// TIA Portal project "Proyecto 4" (V17)
// Clasificador de Cajas

(* hardware
DEVICE "S7-1500/ET200MP station_1"  S7-1500 station
   slot 0: "Rail_0"  Rack  6ES7 590-1***0-0AA0
   slot 1: "PLC_1"  CPU 1515-2 PN  6ES7 515-2AM02-0AB0  V2.9
      slot 3: "CPU display_1"  6ES7591-1BA00-0AA0
      slot 32768: "PROFINET interface_1"  X1
         slot 32769: "Port_1"  X1 P1
         slot 32770: "Port_2"  X1 P2
      slot 33024: "PROFINET interface_2"  X2
         slot 33025: "Port_1"  X2 P1
      slot 34817: "Virtual CP interface port_1"  Virtual CP interface port  Virtual CP interface port
   slot 2: "AI 8xU/I/RTD/TC ST_1"  AI 8xU/I/RTD/TC ST  6ES7 531-7KF00-0AB0  V2.0
   slot 3: "AI 8xU/I/RTD/TC ST_2"  AI 8xU/I/RTD/TC ST  6ES7 531-7KF00-0AB0  V2.0
   slot 4: "AI 8xU/I/RTD/TC ST_3"  AI 8xU/I/RTD/TC ST  6ES7 531-7KF00-0AB0  V2.0
   slot 5: "AI 8xU/I/RTD/TC ST_4"  AI 8xU/I/RTD/TC ST  6ES7 531-7KF00-0AB0  V2.0
   slot 6: "DI 16x24VDC BA_1"  DI 16x24VDC BA  6ES7 521-1BH10-0AA0  V1.0
*)

// ===== PLC "PLC_1"  CPU 1515-2 PN =====

VAR_GLOBAL   // PLC tag table "ED"
   "LAE-High" AT %I0.0 : Bool;
   "LAE-Low" AT %I0.1 : Bool;
   "LAE-Pallet" AT %I0.2 : Bool;
   "SLEN" AT %I0.3 : Bool;
   "SREN" AT %I0.4 : Bool;
   "SLEX" AT %I0.5 : Bool;
   "SREX" AT %I0.6 : Bool;
   "Marcha" AT %I0.7 : Bool;
   "Paro" AT %I1.0 : Bool;
   "Reset" AT %I1.1 : Bool;
   "Seta Emergencia" AT %I1.2 : Bool;
   "SL" AT %I1.3 : Bool;
   "Manual" AT %I1.4 : Bool;
   "Auto" AT %I1.5 : Bool;
END_VAR

VAR_GLOBAL   // PLC tag table "SD"
   "CT-right" AT %Q0.0 : Bool;
   "CT-left" AT %Q0.1 : Bool;
   "CT-Unload" AT %Q0.2 : Bool;
   "CT-Load" AT %Q0.3 : Bool;
   "CE" AT %Q0.4 : Bool;
   "CL" AT %Q0.5 : Bool;
   "CR" AT %Q0.6 : Bool;
   "Emitter" AT %Q0.7 : Bool;
   "Remover left" AT %Q1.0 : Bool;
   "Remover right" AT %Q1.1 : Bool;
   "Start light" AT %Q1.2 : Bool;
   "Stop light" AT %Q1.3 : Bool;
   "Reset light" AT %Q1.4 : Bool;
END_VAR

TYPE "UDT_Cinta"
   STRUCT
      Entradas : Struct
         ParoxSeguridad : Bool;
         Termico : Bool;
         Disyuntor : Bool;
         Auto : Bool;
         ConfMarcha : Bool;
         FalloVariador : Bool;
      END_STRUCT;
      Habilitado : Bool;
      Rearme : Bool;
      HMI : Struct
         Habilitado : Bool;
         segTrabajo : Int;
         minTrabajo : Int;
         horaTrabajo : Int;
      END_STRUCT;
      Alarma : Array[1..16] of Bool;
      AutoRearme : Array[1..16] of Bool;
      TimerAlarma : Array[1..16] of TON_TIME;
      TiempoAlarma : Array[1..16] of Time;
      "Timer" : Array[1..16] of TON_TIME;
      TimerON : Array[1..16] of Bool;
      Salidas : Struct
         Marcha : Bool;
      END_STRUCT;
      Permiso : Struct
         Externo : Bool;
      END_STRUCT;
   END_STRUCT;
END_TYPE

TYPE "UDT_Temporizador"
   STRUCT
      Congelacion : Bool;
      Reset : Bool;
      Q : Bool;
      Tiempo : Int;
      Conteo : Int;
   END_STRUCT;
END_TYPE

TYPE "UDT_Sensor"
   STRUCT
      Value : Bool;
      TON : "UDT_Temporizador";
   END_STRUCT;
END_TYPE

TYPE "UDT_Cinta_Bilateral"
   STRUCT
      Entradas : Struct
         ParoxSeguridad : Bool;
         Termico : Bool;
         Disyuntor : Bool;
         Auto : Bool;
         ConfMarcha : Bool;
         FalloVariador : Bool;
      END_STRUCT;
      Habilitado : Bool;
      Rearme : Bool;
      HMI : Struct
         Habilitado : Bool;
         segTrabajo : Int;
         minTrabajo : Int;
         horaTrabajo : Int;
      END_STRUCT;
      Alarma : Array[1..16] of Bool;
      AutoRearme : Array[1..16] of Bool;
      TimerAlarma : Array[1..16] of TON_TIME;
      TiempoAlarma : Array[1..16] of Time;
      "Timer" : Array[1..16] of TON_TIME;
      TimerON : Array[1..16] of Bool;
      Salidas : Struct
         MarchaAdelante : Bool;
         MarchaAtras : Bool;
         MarchaDch : Bool;
         MarchaIzq : Bool;
      END_STRUCT;
      Permiso : Struct
         Adelante : Bool;
         Atras : Bool;
         Derecha : Bool;
         Izquierda : Bool;
      END_STRUCT;
   END_STRUCT;
END_TYPE

DATA_BLOCK "DB_Generalidades"   // DB1
{ S7_Optimized_Access := 'TRUE' }
VERSION : 0.1
   VAR
      SiempreON : Bool;
      SiempreOFF : Bool;
      Tiempo : Struct
         Imp1ms : Bool;
         Imp1s : Bool;
         Imp1m : Bool;
         Imp1h : Bool;
         TON1ms : TON_TIME;
         TON1s : TON_TIME;
         TON1m : TON_TIME;
         TON1h : TON_TIME;
      END_STRUCT;
   END_VAR
BEGIN
END_DATA_BLOCK

// folder: 01_E/S

DATA_BLOCK "ED"   // DB2
{ S7_Optimized_Access := 'TRUE' }
VERSION : 0.1
   VAR
      "LAE-High" : Bool;
      "LAE-Low" : Bool;
      "LAE-Pallet" : Bool;
      SLEN : Bool;
      SREN : Bool;
      SLEX : Bool;
      SREX : Bool;
      Marcha : Bool;
      Paro : Bool;
      Reset : Bool;
      "Seta Emergencia" : Bool;
      SL : Bool;
      Manual : Bool;
      Auto : Bool;
   END_VAR
BEGIN
END_DATA_BLOCK

DATA_BLOCK "SD"   // DB3
{ S7_Optimized_Access := 'TRUE' }
VERSION : 0.1
   VAR
      "CT-right" : Bool;
      "CT-left" : Bool;
      "CT-Unload" : Bool;
      "CT-Load" : Bool;
      CE : Bool;
      CL : Bool;
      CR : Bool;
      Emitter : Bool;
      "Remover left" : Bool;
      "Remover right" : Bool;
      "Start light" : Bool;
      "Stop light" : Bool;
      "Reset light" : Bool;
   END_VAR
BEGIN
END_DATA_BLOCK

// folder: 02_Equipos

DATA_BLOCK "DB_SensoresDigitales"   // DB100
{ S7_Optimized_Access := 'TRUE' }
VERSION : 0.1
   VAR
      "LAE-High" : "UDT_Sensor";
      "LAE-Low" : "UDT_Sensor";
      "LAE-Pallet" : "UDT_Sensor";
      SLEN : "UDT_Sensor";
      SREN : "UDT_Sensor";
      SREX : "UDT_Sensor";
      SLEX : "UDT_Sensor";
      SetaEmergencia : "UDT_Sensor";
      SL : "UDT_Sensor";
      Paro : "UDT_Sensor";
   END_VAR
BEGIN
END_DATA_BLOCK

DATA_BLOCK "DB_Cintas"   // DB101
{ S7_Optimized_Access := 'TRUE' }
VERSION : 0.1
   VAR
      Unidireccional : Struct
         CE : "UDT_Cinta";
         CL : "UDT_Cinta";
         CR : "UDT_Cinta";
      END_STRUCT;
      Bidireccional : Struct
         CT : "UDT_Cinta_Bilateral";
      END_STRUCT;
   END_VAR
BEGIN
END_DATA_BLOCK

// folder: 10_Zona de Clasificacion

DATA_BLOCK "DB_ZonaClasificacion"   // DB200
{ S7_Optimized_Access := 'TRUE' }
VERSION : 0.1
   VAR
      EnMarcha : Bool;
      EnParo : Bool;
      Flanco : Array[1..32] of Bool;
      CajaEsperando : Bool;
      CajaEnCT : Bool;
      CajaGrande : Bool;
      CajaPequeña : Bool;
      CajaEnCR : Bool;
      CajaEnCL : Bool;
      CajasEnCR : Int;
      CajasEnCL : Int;
   END_VAR
BEGIN
END_DATA_BLOCK

// folder: (top level)

FUNCTION "FC_Generalidades" : Void   // FC1, LAD
{ S7_Optimized_Access := 'TRUE' }
VERSION : 0.1
BEGIN

REGION Network 1: +++++|SIEMPRE ON|+++++
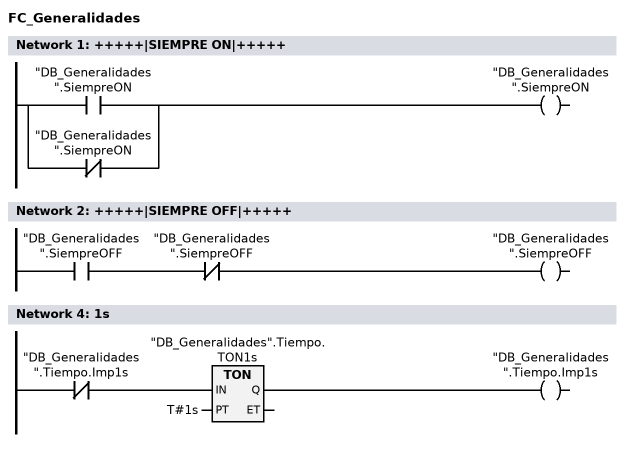
   RUNG wire#powerrail
      Contact( "DB_Generalidades".SiempreON )
      wire#w1
      Coil( "DB_Generalidades".SiempreON )
   END_RUNG
   RUNG wire#powerrail
      I_Contact( "DB_Generalidades".SiempreON )
   END_RUNG wire#w1
   // the same network as SCL:
   "DB_Generalidades".SiempreON := "DB_Generalidades".SiempreON OR NOT "DB_Generalidades".SiempreON;
END_REGION

REGION Network 2: +++++|SIEMPRE OFF|+++++
   RUNG wire#powerrail
      Contact( "DB_Generalidades".SiempreOFF )
      I_Contact( "DB_Generalidades".SiempreOFF )
      Coil( "DB_Generalidades".SiempreOFF )
   END_RUNG
   // the same network as SCL:
   "DB_Generalidades".SiempreOFF := "DB_Generalidades".SiempreOFF AND NOT "DB_Generalidades".SiempreOFF;
END_REGION

REGION Network 3: +++++|IMPULSOS DE TIEMPO|+++++
END_REGION

REGION Network 4: 1s
   "DB_Generalidades".Tiempo.TON1s.TON(IN := NOT "DB_Generalidades".Tiempo.Imp1s, PT := T#1s);
   "DB_Generalidades".Tiempo.Imp1s := "DB_Generalidades".Tiempo.TON1s.Q;
END_REGION
END_FUNCTION

FUNCTION "MHJ-PLC-Lab-Function-S71500" : Void   // FC9000, SCL
{ S7_Optimized_Access := 'TRUE' }
VERSION : 0.1
   VAR_TEMP
      Value : Byte;
      ForCounter : Int;
   END_VAR
   VAR CONSTANT
      Value_01_DW : DWord := 16#1223_5486;
      Value_02_DW : DWord := 16#A6C9_D1F5;
   END_VAR
BEGIN

   #Value:=PEEK(area := 16#82,
        dbNumber := 0,
        byteOffset := 511);
   #Value := #Value + 1;

   POKE(area := 16#82,
        dbNumber := 0,
        byteOffset := 511,
        value := #Value);

   POKE(area := 16#82,
        dbNumber := 0,
        byteOffset := 1016,
        value := #Value_01_DW);
   POKE(area := 16#82,
        dbNumber := 0,
        byteOffset := 1020,
        value := #Value_02_DW);

   FOR #ForCounter := 0 TO 63 DO
       #Value:=PEEK(area := 16#1,
            dbNumber := 0,
            byteOffset := #ForCounter);
       POKE(area := 16#81,
            dbNumber := 0,
            byteOffset := #ForCounter,
            value := #Value);
   END_FOR;
   #Value := PEEK(area := 16#1,
                  dbNumber := 0,
                  byteOffset := 512);
   POKE(area := 16#82,
        dbNumber := 0,
        byteOffset := 512,
        value := #Value);
END_FUNCTION

ORGANIZATION_BLOCK "Main"   // OB1, LAD, ProgramCycle
TITLE = "Main Program Sweep (Cycle)"
{ S7_Optimized_Access := 'TRUE' }
VERSION : 0.1
// BENONI BENJAMIN QUEZADA FLORES
   VAR_INPUT
      Initial_Call : Bool;   // Initial call of this OB
      Remanence : Bool;   // =True, if remanent data are available
   END_VAR
BEGIN

REGION Network 1 (STL): +++++|LECTURA ENTRADAS|+++++

         CALL  "FC_ED";
END_REGION

REGION Network 2 (STL): +++++|GENERALIDADES|+++++

         CALL  "FC_Generalidades";
END_REGION

REGION Network 3 (STL): +++++|COMUNICACION FACTORY IO|+++++

         CALL  "MHJ-PLC-Lab-Function-S71500";
END_REGION

REGION Network 4 (STL): +++++|ZONA CLASIFICACION|+++++

         CALL  "FC_ZonaClasificacion";
END_REGION

REGION Network 5 (STL): +++++|ESCRITURAS SALIDAS|+++++

         CALL  "FC_SD";
END_REGION
END_ORGANIZATION_BLOCK

// folder: 00_Bloques Estandar/FB

FUNCTION_BLOCK "FB_Motor"   // FB1, LAD
{ S7_Optimized_Access := 'TRUE' }
VERSION : 0.1
   VAR_INPUT
      eParoXSeguridad : Bool;
      eTermico : Bool;
      eDisyuntor : Bool;
      eAuto : Bool;
      eConfMarcha : Bool;
      eFalloVariador : Bool;
   END_VAR
   VAR_OUTPUT
      sMarcha : Bool;
   END_VAR
   VAR
      Habilitado : Bool;
      Rearme : Bool;
      PermisoExterno : Bool;
      HMI : Struct
         Habilitado : Bool;
         segTrabajo : Int;
         minTrabajo : Int;
         horaTrabajo : Int;
      END_STRUCT;
      Alarma : Array[1..16] of Bool;
      AutoRearme : Array[1..16] of Bool;
      TimerAlarma : Array[1..16] of TON_TIME;
      TiempoAlarma : Array[1..16] of Time;
      "Timer" : Array[1..16] of TON_TIME;
      TimerON : Array[1..16] of Bool;
   END_VAR
   VAR_TEMP
      OkAlarma : Bool;
      EnMarcha : Bool;
   END_VAR
BEGIN

REGION Network 1: +++++|Habilitado Motor|+++++
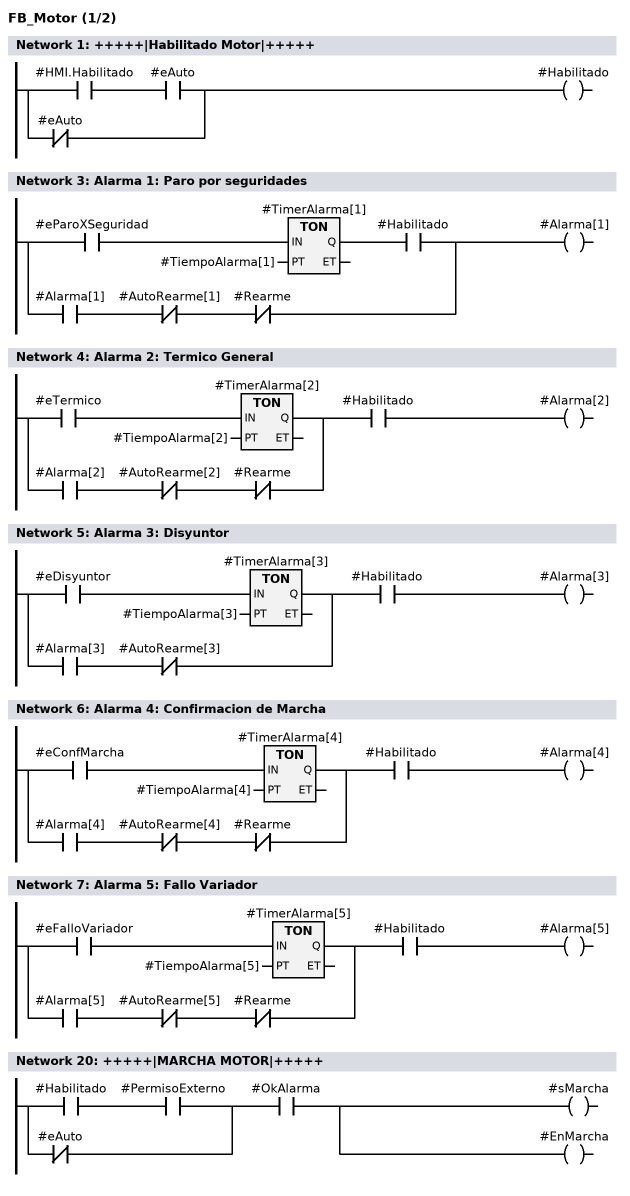
   RUNG wire#powerrail
      Contact( #HMI.Habilitado )
      Contact( #eAuto )
      wire#w1
      Coil( #Habilitado )
   END_RUNG
   RUNG wire#powerrail
      I_Contact( #eAuto )
   END_RUNG wire#w1
   // the same network as SCL:
   #Habilitado := (#HMI.Habilitado AND #eAuto) OR NOT #eAuto;
END_REGION

REGION Network 2: +++++|ALARMAS|+++++
END_REGION

REGION Network 3: Alarma 1: Paro por seguridades
   #TimerAlarma[1].TON(IN := #eParoXSeguridad, PT := #TiempoAlarma[1]);
   #Alarma[1] := (#TimerAlarma[1].Q AND #Habilitado) OR (#Alarma[1] AND NOT #AutoRearme[1] AND NOT #Rearme);
END_REGION

REGION Network 4: Alarma 2: Termico General
   #TimerAlarma[2].TON(IN := #eTermico, PT := #TiempoAlarma[2]);
   #Alarma[2] := (#TimerAlarma[2].Q OR (#Alarma[2] AND NOT #AutoRearme[2] AND NOT #Rearme)) AND #Habilitado;
END_REGION

REGION Network 5: Alarma 3: Disyuntor
   #TimerAlarma[3].TON(IN := #eDisyuntor, PT := #TiempoAlarma[3]);
   #Alarma[3] := (#TimerAlarma[3].Q OR (#Alarma[3] AND NOT #AutoRearme[3])) AND #Habilitado;
END_REGION

REGION Network 6: Alarma 4: Confirmacion de Marcha
   #TimerAlarma[4].TON(IN := #eConfMarcha, PT := #TiempoAlarma[4]);
   #Alarma[4] := (#TimerAlarma[4].Q OR (#Alarma[4] AND NOT #AutoRearme[4] AND NOT #Rearme)) AND #Habilitado;
END_REGION

REGION Network 7: Alarma 5: Fallo Variador
   #TimerAlarma[5].TON(IN := #eFalloVariador, PT := #TiempoAlarma[5]);
   #Alarma[5] := (#TimerAlarma[5].Q OR (#Alarma[5] AND NOT #AutoRearme[5] AND NOT #Rearme)) AND #Habilitado;
END_REGION

REGION Network 8: Alarma 6: Reserva
END_REGION

REGION Network 9: Alarma 7: Reserva
END_REGION

REGION Network 10: Alarma 8:Reserva
END_REGION

REGION Network 11: Alarma 9: Reserva
END_REGION

REGION Network 12: Alarma 10:Reserva
END_REGION

REGION Network 13: Alarma 11: Reserva
END_REGION

REGION Network 14: Alarma 12: Reserva
END_REGION

REGION Network 15: Alarma 13: Reserva
END_REGION

REGION Network 16: Alarma 14: Reserva
END_REGION

REGION Network 17: Alarma 15: Reserva
END_REGION

REGION Network 18: Alarma 16: Reserva
END_REGION

REGION Network 19 (STL): +++++|RESUMEN ALARMAS|+++++
         AN    #Alarma[1];
         AN    #Alarma[2];
         AN    #Alarma[3];
         AN    #Alarma[4];
         AN    #Alarma[5];
         AN    #Alarma[6];
         AN    #Alarma[7];
         AN    #Alarma[8];
         AN    #Alarma[9];
         AN    #Alarma[10];
         AN    #Alarma[11];
         AN    #Alarma[12];
         AN    #Alarma[13];
         AN    #Alarma[14];
         AN    #Alarma[15];
         AN    #Alarma[16];
         =     #OkAlarma;
END_REGION

REGION Network 20: +++++|MARCHA MOTOR|+++++
   RUNG wire#powerrail
      Contact( #Habilitado )
      Contact( #PermisoExterno )
      wire#w1
      Contact( #OkAlarma )
      wire#w2
      Coil( #sMarcha )
   END_RUNG
   RUNG wire#powerrail
      I_Contact( #eAuto )
   END_RUNG wire#w1
   RUNG wire#w2
      Coil( #EnMarcha )
   END_RUNG
   // the same network as SCL:
   #sMarcha := ((#Habilitado AND #PermisoExterno) OR NOT #eAuto) AND #OkAlarma;
   #EnMarcha := #sMarcha;
END_REGION

REGION Network 21: +++++|TIEMPO DE TRABAJO|+++++
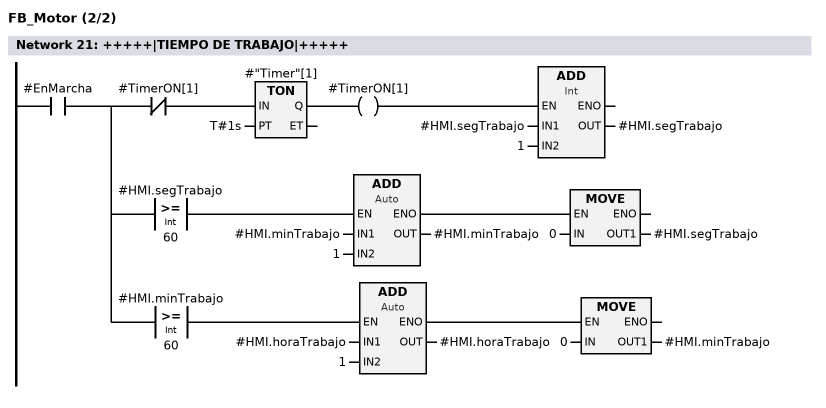
   #"Timer"[1].TON(IN := #EnMarcha AND NOT #TimerON[1], PT := T#1s);
   #TimerON[1] := #"Timer"[1].Q;
   IF #"Timer"[1].Q THEN #HMI.segTrabajo := #HMI.segTrabajo + 1; END_IF;
   IF #EnMarcha AND (#HMI.segTrabajo >= 60) THEN
       #HMI.minTrabajo := #HMI.minTrabajo + 1;
       #HMI.segTrabajo := 0;
   END_IF;
   IF #EnMarcha AND (#HMI.minTrabajo >= 60) THEN
       #HMI.horaTrabajo := #HMI.horaTrabajo + 1;
       #HMI.minTrabajo := 0;
   END_IF;
END_REGION
END_FUNCTION_BLOCK

// folder: 00_Bloques Estandar/FC/00_Utilidades

FUNCTION "TOFF" : Void   // FC4, LAD
TITLE = +++++|TEMPORIZADOR DESCENDENTE|+++++
{ S7_Optimized_Access := 'TRUE' }
VERSION : 0.1
   VAR_INPUT
      Activacion : Bool;
      Impulso : Bool;   // ms,s,min,h
      Congelacion : Bool;
      Reset : Bool;
      Tiempo : Int;
   END_VAR
   VAR_IN_OUT
      Conteo : Int;
      Q : Bool;
   END_VAR
   VAR_TEMP   // added for the SCL form of the ladder/FBD networks
      _w1 : Bool;
   END_VAR
BEGIN

REGION Network 1: +++++|ACTIVACION|+++++
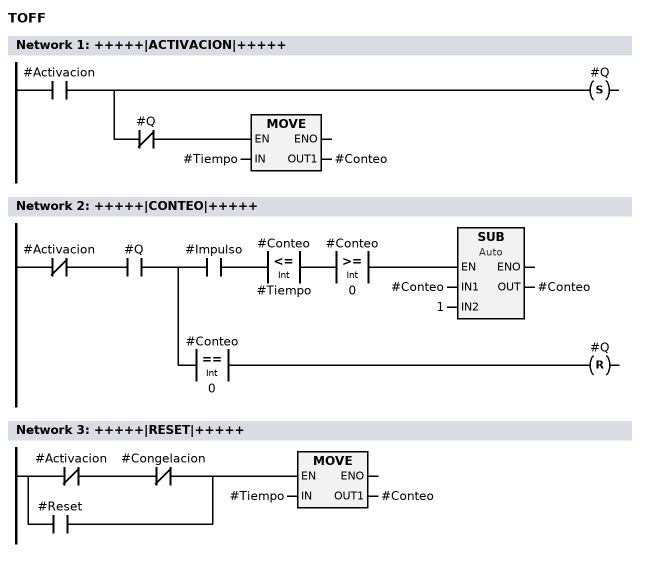
   RUNG wire#powerrail
      Contact( #Activacion )
      wire#w1
      S_Coil( #Q )
   END_RUNG
   RUNG wire#w1
      I_Contact( #Q )
      Move(in := #Tiempo, out1 => #Conteo)
   END_RUNG
   // the same network as SCL:
   IF #Activacion THEN #Q := TRUE; END_IF;
   IF #Activacion AND NOT #Q THEN #Conteo := #Tiempo; END_IF;
END_REGION

REGION Network 2: +++++|CONTEO|+++++
   RUNG wire#powerrail
      I_Contact( #Activacion )
      Contact( #Q )
      wire#w1
      Contact( #Impulso )
      { S7_Templates := "SrcType := Int" } LE_Contact(in1 := #Conteo, in2 := #Tiempo)
      { S7_Templates := "SrcType := Int" } GE_Contact(in1 := #Conteo, in2 := 0)
      Sub(in1 := #Conteo, in2 := 1, out => #Conteo)
   END_RUNG
   RUNG wire#w1
      { S7_Templates := "SrcType := Int" } EQ_Contact(in1 := #Conteo, in2 := 0)
      R_Coil( #Q )
   END_RUNG
   // the same network as SCL:
   #_w1 := NOT #Activacion AND #Q;
   IF #_w1 AND #Impulso AND (#Conteo <= #Tiempo) AND (#Conteo >= 0) THEN #Conteo := #Conteo - 1; END_IF;
   IF #_w1 AND (#Conteo = 0) THEN #Q := FALSE; END_IF;
END_REGION

REGION Network 3: +++++|RESET|+++++
   RUNG wire#powerrail
      I_Contact( #Activacion )
      I_Contact( #Congelacion )
      wire#w1
      Move(in := #Tiempo, out1 => #Conteo)
   END_RUNG
   RUNG wire#powerrail
      Contact( #Reset )
   END_RUNG wire#w1
   // the same network as SCL:
   IF (NOT #Activacion AND NOT #Congelacion) OR #Reset THEN #Conteo := #Tiempo; END_IF;
END_REGION

REGION Network 4 (STL): +++++|ACTIVACION SALIDA MEDIANTE EN0|+++++
         A     #Q;
         SAVE;
END_REGION
END_FUNCTION

FUNCTION "TON" : Void   // FC10, LAD
{ S7_Optimized_Access := 'TRUE' }
VERSION : 0.1
   VAR_INPUT
      Activacion : Bool;
      Impulso : Bool;   // ms,s,min,h
      Congelacion : Bool;
      Reset : Bool;
      Tiempo : Int;
   END_VAR
   VAR_IN_OUT
      Conteo : Int;
   END_VAR
   VAR_TEMP
      Q : Bool;
   END_VAR
BEGIN

REGION Network 1: +++++|TEMPORIZADOR ASCENDENTE|+++++
END_REGION

REGION Network 2: +++++|ACTIVACION|+++++
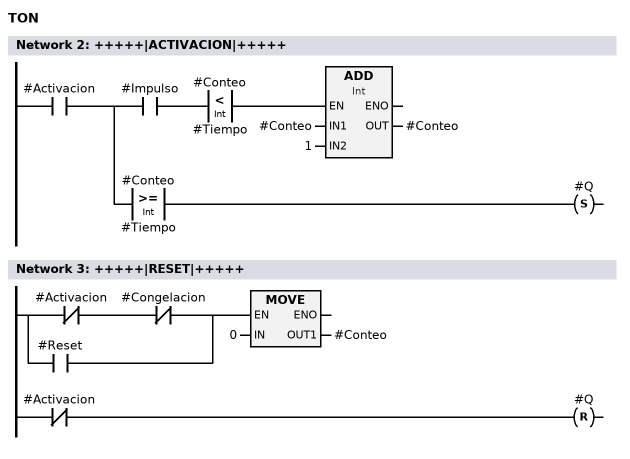
   RUNG wire#powerrail
      Contact( #Activacion )
      wire#w1
      Contact( #Impulso )
      { S7_Templates := "SrcType := Int" } LT_Contact(in1 := #Conteo, in2 := #Tiempo)
      { S7_Templates := "SrcType := Int" } Add(in1 := #Conteo, in2 := 1, out => #Conteo)
   END_RUNG
   RUNG wire#w1
      { S7_Templates := "SrcType := Int" } GE_Contact(in1 := #Conteo, in2 := #Tiempo)
      S_Coil( #Q )
   END_RUNG
   // the same network as SCL:
   IF #Activacion AND #Impulso AND (#Conteo < #Tiempo) THEN #Conteo := #Conteo + 1; END_IF;
   IF #Activacion AND (#Conteo >= #Tiempo) THEN #Q := TRUE; END_IF;
END_REGION

REGION Network 3: +++++|RESET|+++++
   RUNG wire#powerrail
      I_Contact( #Activacion )
      I_Contact( #Congelacion )
      wire#w1
      Move(in := 0, out1 => #Conteo)
   END_RUNG
   RUNG wire#powerrail
      Contact( #Reset )
   END_RUNG wire#w1
   RUNG wire#powerrail
      I_Contact( #Activacion )
      R_Coil( #Q )
   END_RUNG
   // the same network as SCL:
   IF (NOT #Activacion AND NOT #Congelacion) OR #Reset THEN #Conteo := 0; END_IF;
   IF NOT #Activacion THEN #Q := FALSE; END_IF;
END_REGION

REGION Network 4 (STL): +++++|ACTIVACION SALIDA MEDIANTE EN0|+++++
         A     #Q;
         SAVE;
END_REGION
END_FUNCTION

// folder: 00_Bloques Estandar/FC/01_Equipos

FUNCTION "FC_SensorDigital" : Void   // FC100, LAD
TITLE = +++++|TRATAMIENTO SENSOR DIGITAL|+++++
{ S7_Optimized_Access := 'TRUE' }
VERSION : 0.1
   VAR_INPUT
      Sensor : Bool;
      Negado : Bool;
      Retardo : Int;
   END_VAR
   VAR_IN_OUT
      UDT_Sensor : "UDT_Sensor";
   END_VAR
   VAR_TEMP
      Activado : Bool;
   END_VAR
   VAR_TEMP   // added for the SCL form of the ladder/FBD networks
      _w1 : Bool;
   END_VAR
BEGIN

REGION Network 1: Configuracion Segun la logica de funcionamiento
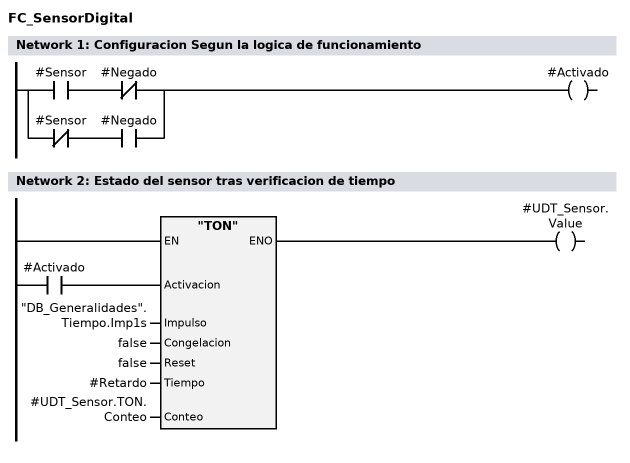
   RUNG wire#powerrail
      Contact( #Sensor )
      I_Contact( #Negado )
      wire#w1
      Coil( #Activado )
   END_RUNG
   RUNG wire#powerrail
      I_Contact( #Sensor )
      Contact( #Negado )
   END_RUNG wire#w1
   // the same network as SCL:
   #Activado := (#Sensor AND NOT #Negado) OR (NOT #Sensor AND #Negado);
END_REGION

REGION Network 2: Estado del sensor tras verificacion de tiempo
   RUNG wire#powerrail
      "TON"(Activacion := wire#w1, Impulso := "DB_Generalidades".Tiempo.Imp1s, Congelacion := false, Reset := false, Tiempo := #Retardo, Conteo := #UDT_Sensor.TON.Conteo)
      Coil( #UDT_Sensor.Value )
   END_RUNG
   RUNG wire#powerrail
      Contact( #Activado )
   END_RUNG wire#w1
   // the same network as SCL:
   "TON"(Activacion := #Activado,
         Impulso := "DB_Generalidades".Tiempo.Imp1s,
         Congelacion := false,
         Reset := false,
         Tiempo := #Retardo,
         Conteo := #UDT_Sensor.TON.Conteo,
         ENO => #_w1);
   #UDT_Sensor.Value := #_w1;
END_REGION
END_FUNCTION

FUNCTION "FC_Cinta" : Void   // FC101, LAD
TITLE = Cinta Transportadora
{ S7_Optimized_Access := 'TRUE' }
VERSION : 0.1
   VAR_IN_OUT
      Cinta : "UDT_Cinta";
   END_VAR
   VAR_TEMP
      OkAlarma : Bool;
      EnMarcha : Bool;
   END_VAR
BEGIN

REGION Network 1: +++++|HABILITAR CINTA|+++++
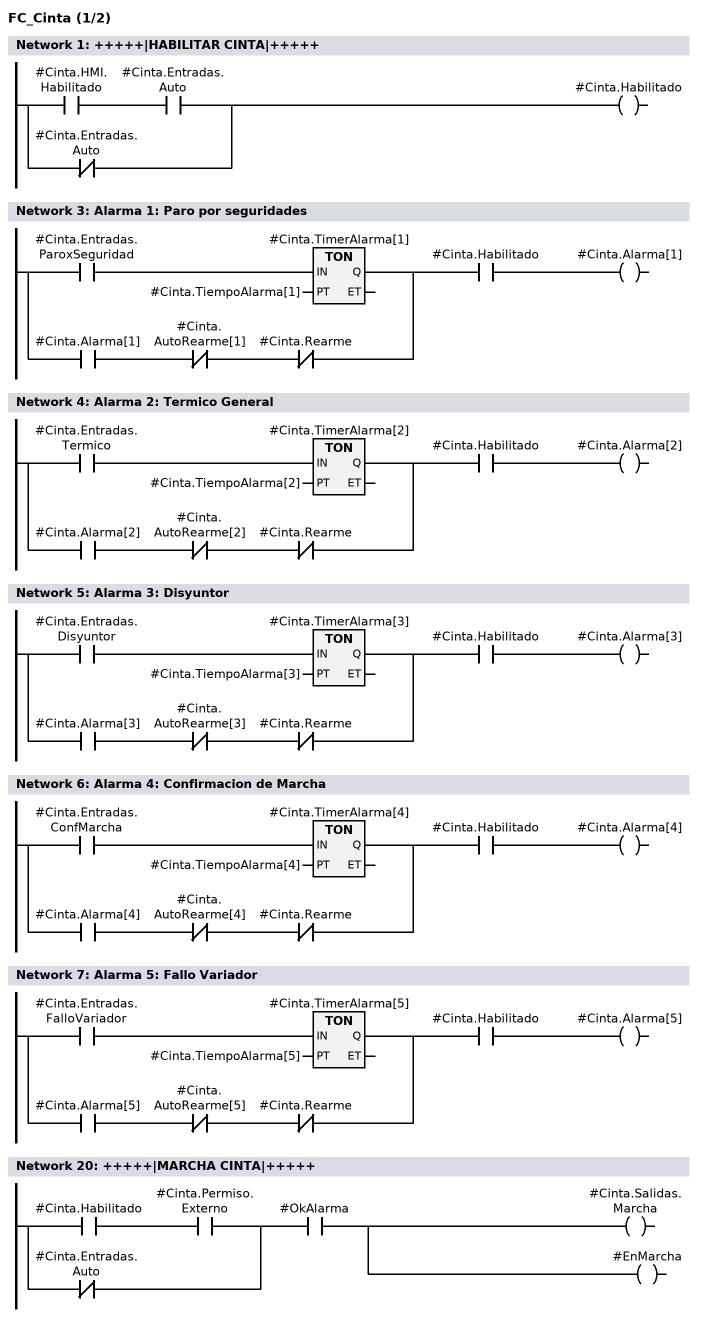
   RUNG wire#powerrail
      Contact( #Cinta.HMI.Habilitado )
      Contact( #Cinta.Entradas.Auto )
      wire#w1
      Coil( #Cinta.Habilitado )
   END_RUNG
   RUNG wire#powerrail
      I_Contact( #Cinta.Entradas.Auto )
   END_RUNG wire#w1
   // the same network as SCL:
   #Cinta.Habilitado := (#Cinta.HMI.Habilitado AND #Cinta.Entradas.Auto) OR NOT #Cinta.Entradas.Auto;
END_REGION

REGION Network 2: +++++|ALARMAS|+++++
END_REGION

REGION Network 3: Alarma 1: Paro por seguridades
   #Cinta.TimerAlarma[1].TON(IN := #Cinta.Entradas.ParoxSeguridad, PT := #Cinta.TiempoAlarma[1]);
   #Cinta.Alarma[1] := (#Cinta.TimerAlarma[1].Q OR (#Cinta.Alarma[1] AND NOT #Cinta.AutoRearme[1] AND NOT #Cinta.Rearme)) AND #Cinta.Habilitado;
END_REGION

REGION Network 4: Alarma 2: Termico General
   #Cinta.TimerAlarma[2].TON(IN := #Cinta.Entradas.Termico, PT := #Cinta.TiempoAlarma[2]);
   #Cinta.Alarma[2] := (#Cinta.TimerAlarma[2].Q OR (#Cinta.Alarma[2] AND NOT #Cinta.AutoRearme[2] AND NOT #Cinta.Rearme)) AND #Cinta.Habilitado;
END_REGION

REGION Network 5: Alarma 3: Disyuntor
   #Cinta.TimerAlarma[3].TON(IN := #Cinta.Entradas.Disyuntor, PT := #Cinta.TiempoAlarma[3]);
   #Cinta.Alarma[3] := (#Cinta.TimerAlarma[3].Q OR (#Cinta.Alarma[3] AND NOT #Cinta.AutoRearme[3] AND NOT #Cinta.Rearme)) AND #Cinta.Habilitado;
END_REGION

REGION Network 6: Alarma 4: Confirmacion de Marcha
   #Cinta.TimerAlarma[4].TON(IN := #Cinta.Entradas.ConfMarcha, PT := #Cinta.TiempoAlarma[4]);
   #Cinta.Alarma[4] := (#Cinta.TimerAlarma[4].Q OR (#Cinta.Alarma[4] AND NOT #Cinta.AutoRearme[4] AND NOT #Cinta.Rearme)) AND #Cinta.Habilitado;
END_REGION

REGION Network 7: Alarma 5: Fallo Variador
   #Cinta.TimerAlarma[5].TON(IN := #Cinta.Entradas.FalloVariador, PT := #Cinta.TiempoAlarma[5]);
   #Cinta.Alarma[5] := (#Cinta.TimerAlarma[5].Q OR (#Cinta.Alarma[5] AND NOT #Cinta.AutoRearme[5] AND NOT #Cinta.Rearme)) AND #Cinta.Habilitado;
END_REGION

REGION Network 8: Alarma 6: Reserva
END_REGION

REGION Network 9: Alarma 7: Reserva
END_REGION

REGION Network 10: Alarma 8: Reserva
END_REGION

REGION Network 11: Alarma 9: Reserva
END_REGION

REGION Network 12: Alarma 10: Reserva
END_REGION

REGION Network 13: Alarma 11: Reserva
END_REGION

REGION Network 14: Alarma 12: Reserva
END_REGION

REGION Network 15: Alarma 13: Reserva
END_REGION

REGION Network 16: Alarma 14: Reserva
END_REGION

REGION Network 17: Alarma 15: Reserva
END_REGION

REGION Network 18: Alarma 16: Reserva
END_REGION

REGION Network 19 (STL): +++++|RESUMEN ALARMAS|+++++
         AN    #Cinta.Alarma[1];
         AN    #Cinta.Alarma[2];
         AN    #Cinta.Alarma[3];
         AN    #Cinta.Alarma[4];
         AN    #Cinta.Alarma[5];
         AN    #Cinta.Alarma[6];
         AN    #Cinta.Alarma[7];
         AN    #Cinta.Alarma[8];
         AN    #Cinta.Alarma[9];
         AN    #Cinta.Alarma[10];
         AN    #Cinta.Alarma[11];
         AN    #Cinta.Alarma[12];
         AN    #Cinta.Alarma[13];
         AN    #Cinta.Alarma[14];
         AN    #Cinta.Alarma[15];
         AN    #Cinta.Alarma[16];
         =     #OkAlarma;
END_REGION

REGION Network 20: +++++|MARCHA CINTA|+++++
   RUNG wire#powerrail
      Contact( #Cinta.Habilitado )
      Contact( #Cinta.Permiso.Externo )
      wire#w1
      Contact( #OkAlarma )
      wire#w2
      Coil( #Cinta.Salidas.Marcha )
   END_RUNG
   RUNG wire#powerrail
      I_Contact( #Cinta.Entradas.Auto )
   END_RUNG wire#w1
   RUNG wire#w2
      Coil( #EnMarcha )
   END_RUNG
   // the same network as SCL:
   #Cinta.Salidas.Marcha := ((#Cinta.Habilitado AND #Cinta.Permiso.Externo) OR NOT #Cinta.Entradas.Auto) AND #OkAlarma;
   #EnMarcha := #Cinta.Salidas.Marcha;
END_REGION

REGION Network 21: +++++|TIEMPO DE TRABAJO|+++++
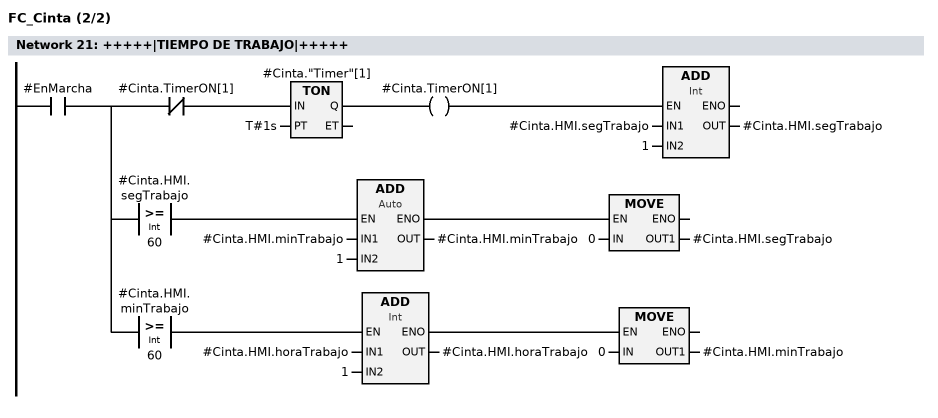
   #Cinta."Timer"[1].TON(IN := #EnMarcha AND NOT #Cinta.TimerON[1], PT := T#1s);
   #Cinta.TimerON[1] := #Cinta."Timer"[1].Q;
   IF #Cinta."Timer"[1].Q THEN #Cinta.HMI.segTrabajo := #Cinta.HMI.segTrabajo + 1; END_IF;
   IF #EnMarcha AND (#Cinta.HMI.segTrabajo >= 60) THEN
       #Cinta.HMI.minTrabajo := #Cinta.HMI.minTrabajo + 1;
       #Cinta.HMI.segTrabajo := 0;
   END_IF;
   IF #EnMarcha AND (#Cinta.HMI.minTrabajo >= 60) THEN
       #Cinta.HMI.horaTrabajo := #Cinta.HMI.horaTrabajo + 1;
       #Cinta.HMI.minTrabajo := 0;
   END_IF;
END_REGION
END_FUNCTION

FUNCTION "FC_Cinta_Bidireccional" : Void   // FC102, LAD
TITLE = Cinta Transportadora Bilateral
{ S7_Optimized_Access := 'TRUE' }
VERSION : 0.1
   VAR_IN_OUT
      Cinta : "UDT_Cinta_Bilateral";
   END_VAR
   VAR_TEMP
      OkAlarma : Bool;
      EnMarcha : Bool;
   END_VAR
BEGIN

REGION Network 1: +++++|HABILITAR CINTA|+++++
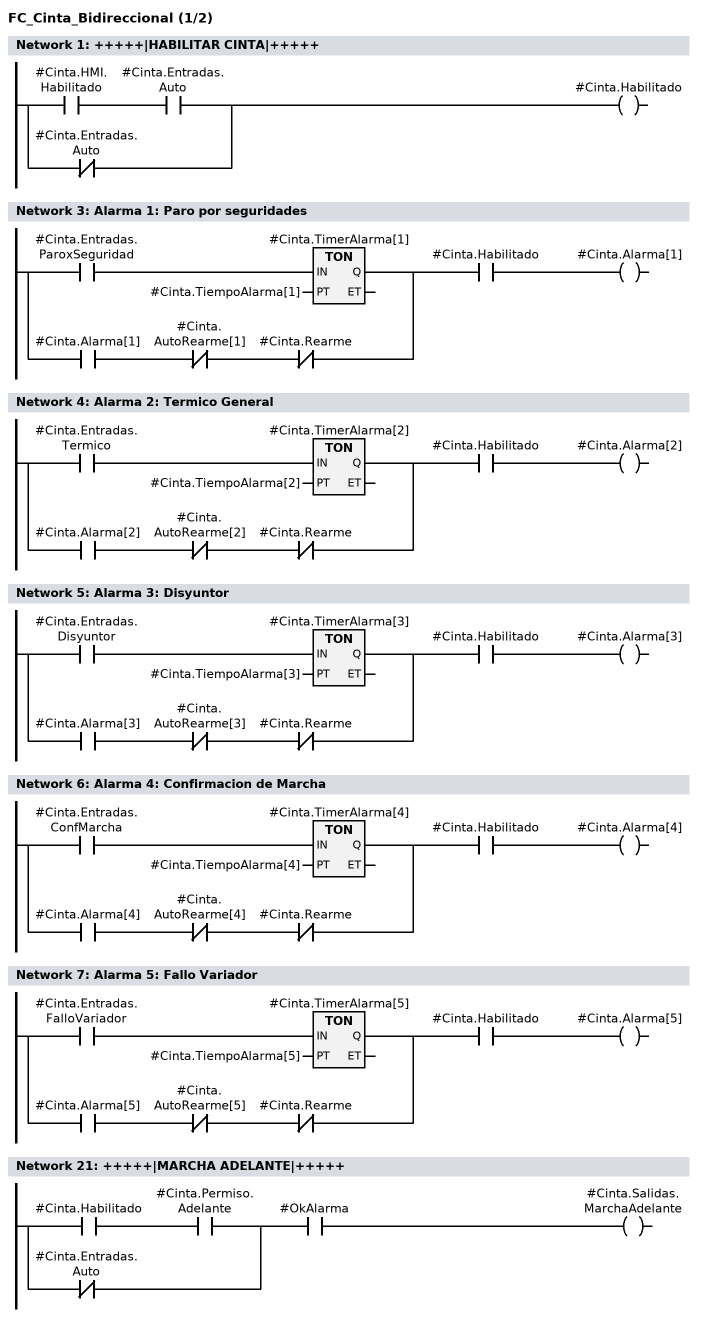
   RUNG wire#powerrail
      Contact( #Cinta.HMI.Habilitado )
      Contact( #Cinta.Entradas.Auto )
      wire#w1
      Coil( #Cinta.Habilitado )
   END_RUNG
   RUNG wire#powerrail
      I_Contact( #Cinta.Entradas.Auto )
   END_RUNG wire#w1
   // the same network as SCL:
   #Cinta.Habilitado := (#Cinta.HMI.Habilitado AND #Cinta.Entradas.Auto) OR NOT #Cinta.Entradas.Auto;
END_REGION

REGION Network 2: +++++|ALARMAS|+++++
END_REGION

REGION Network 3: Alarma 1: Paro por seguridades
   #Cinta.TimerAlarma[1].TON(IN := #Cinta.Entradas.ParoxSeguridad, PT := #Cinta.TiempoAlarma[1]);
   #Cinta.Alarma[1] := (#Cinta.TimerAlarma[1].Q OR (#Cinta.Alarma[1] AND NOT #Cinta.AutoRearme[1] AND NOT #Cinta.Rearme)) AND #Cinta.Habilitado;
END_REGION

REGION Network 4: Alarma 2: Termico General
   #Cinta.TimerAlarma[2].TON(IN := #Cinta.Entradas.Termico, PT := #Cinta.TiempoAlarma[2]);
   #Cinta.Alarma[2] := (#Cinta.TimerAlarma[2].Q OR (#Cinta.Alarma[2] AND NOT #Cinta.AutoRearme[2] AND NOT #Cinta.Rearme)) AND #Cinta.Habilitado;
END_REGION

REGION Network 5: Alarma 3: Disyuntor
   #Cinta.TimerAlarma[3].TON(IN := #Cinta.Entradas.Disyuntor, PT := #Cinta.TiempoAlarma[3]);
   #Cinta.Alarma[3] := (#Cinta.TimerAlarma[3].Q OR (#Cinta.Alarma[3] AND NOT #Cinta.AutoRearme[3] AND NOT #Cinta.Rearme)) AND #Cinta.Habilitado;
END_REGION

REGION Network 6: Alarma 4: Confirmacion de Marcha
   #Cinta.TimerAlarma[4].TON(IN := #Cinta.Entradas.ConfMarcha, PT := #Cinta.TiempoAlarma[4]);
   #Cinta.Alarma[4] := (#Cinta.TimerAlarma[4].Q OR (#Cinta.Alarma[4] AND NOT #Cinta.AutoRearme[4] AND NOT #Cinta.Rearme)) AND #Cinta.Habilitado;
END_REGION

REGION Network 7: Alarma 5: Fallo Variador
   #Cinta.TimerAlarma[5].TON(IN := #Cinta.Entradas.FalloVariador, PT := #Cinta.TiempoAlarma[5]);
   #Cinta.Alarma[5] := (#Cinta.TimerAlarma[5].Q OR (#Cinta.Alarma[5] AND NOT #Cinta.AutoRearme[5] AND NOT #Cinta.Rearme)) AND #Cinta.Habilitado;
END_REGION

REGION Network 8: Alarma 6: Reserva
END_REGION

REGION Network 9: Alarma 7: Reserva
END_REGION

REGION Network 10: Alarma 8: Reserva
END_REGION

REGION Network 11: Alarma 9: Reserva
END_REGION

REGION Network 12: Alarma 10: Reserva
END_REGION

REGION Network 13: Alarma 11: Reserva
END_REGION

REGION Network 14: Alarma 12: Reserva
END_REGION

REGION Network 15: Alarma 13: Reserva
END_REGION

REGION Network 16: Alarma 14: Reserva
END_REGION

REGION Network 17: Alarma 15: Reserva
END_REGION

REGION Network 18: Alarma 16: Reserva
END_REGION

REGION Network 19 (STL): +++++|RESUMEN ALARMAS|+++++
         AN    #Cinta.Alarma[1];
         AN    #Cinta.Alarma[2];
         AN    #Cinta.Alarma[3];
         AN    #Cinta.Alarma[4];
         AN    #Cinta.Alarma[5];
         AN    #Cinta.Alarma[6];
         AN    #Cinta.Alarma[7];
         AN    #Cinta.Alarma[8];
         AN    #Cinta.Alarma[9];
         AN    #Cinta.Alarma[10];
         AN    #Cinta.Alarma[11];
         AN    #Cinta.Alarma[12];
         AN    #Cinta.Alarma[13];
         AN    #Cinta.Alarma[14];
         AN    #Cinta.Alarma[15];
         AN    #Cinta.Alarma[16];
         =     #OkAlarma;
END_REGION

REGION Network 20: +++++|MARCHA CINTA|+++++
END_REGION

REGION Network 21: +++++|MARCHA ADELANTE|+++++
   RUNG wire#powerrail
      Contact( #Cinta.Habilitado )
      Contact( #Cinta.Permiso.Adelante )
      wire#w1
      Contact( #OkAlarma )
      Coil( #Cinta.Salidas.MarchaAdelante )
   END_RUNG
   RUNG wire#powerrail
      I_Contact( #Cinta.Entradas.Auto )
   END_RUNG wire#w1
   // the same network as SCL:
   #Cinta.Salidas.MarchaAdelante := ((#Cinta.Habilitado AND #Cinta.Permiso.Adelante) OR NOT #Cinta.Entradas.Auto) AND #OkAlarma;
END_REGION

REGION Network 22: +++++|MARCHA ATRAS|+++++
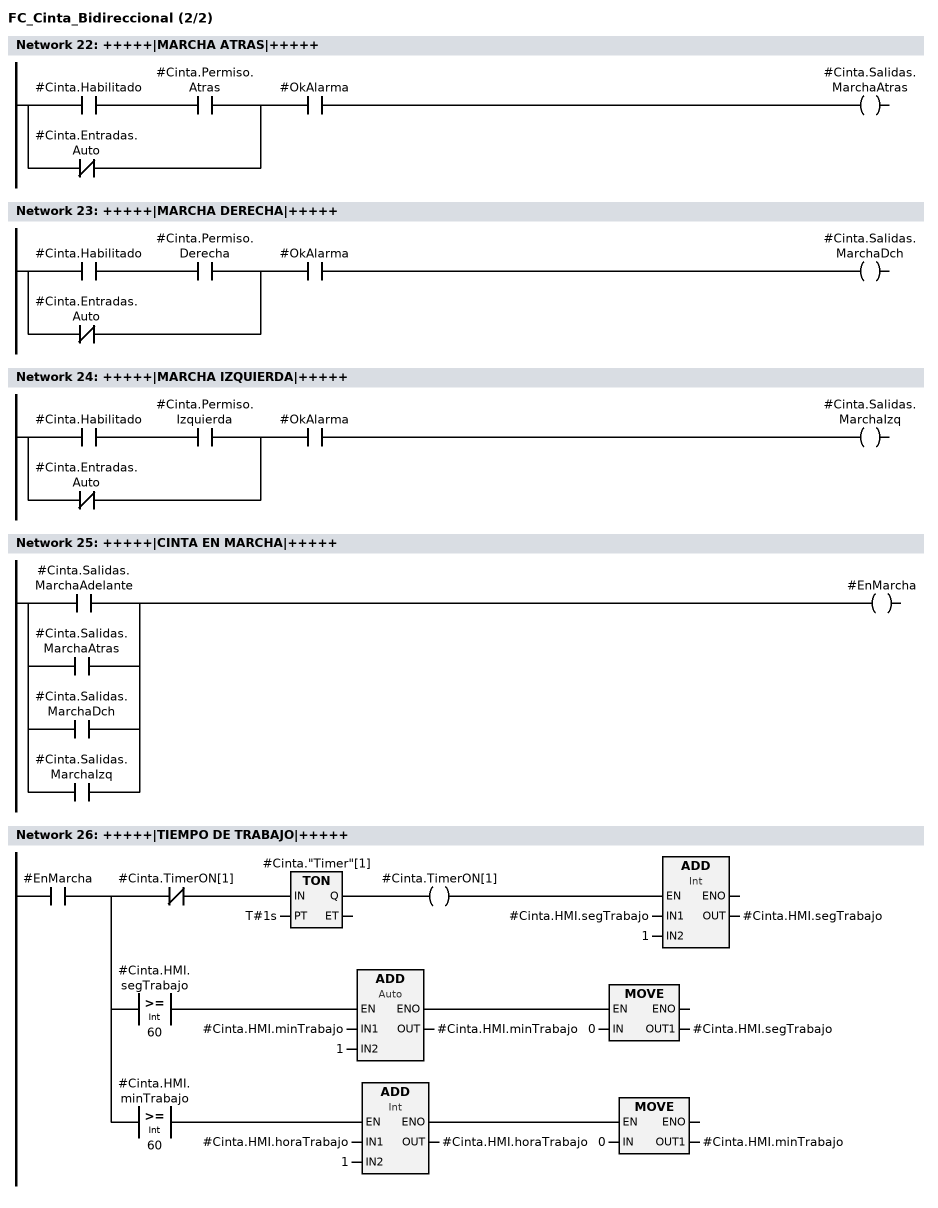
   RUNG wire#powerrail
      Contact( #Cinta.Habilitado )
      Contact( #Cinta.Permiso.Atras )
      wire#w1
      Contact( #OkAlarma )
      Coil( #Cinta.Salidas.MarchaAtras )
   END_RUNG
   RUNG wire#powerrail
      I_Contact( #Cinta.Entradas.Auto )
   END_RUNG wire#w1
   // the same network as SCL:
   #Cinta.Salidas.MarchaAtras := ((#Cinta.Habilitado AND #Cinta.Permiso.Atras) OR NOT #Cinta.Entradas.Auto) AND #OkAlarma;
END_REGION

REGION Network 23: +++++|MARCHA DERECHA|+++++
   RUNG wire#powerrail
      Contact( #Cinta.Habilitado )
      Contact( #Cinta.Permiso.Derecha )
      wire#w1
      Contact( #OkAlarma )
      Coil( #Cinta.Salidas.MarchaDch )
   END_RUNG
   RUNG wire#powerrail
      I_Contact( #Cinta.Entradas.Auto )
   END_RUNG wire#w1
   // the same network as SCL:
   #Cinta.Salidas.MarchaDch := ((#Cinta.Habilitado AND #Cinta.Permiso.Derecha) OR NOT #Cinta.Entradas.Auto) AND #OkAlarma;
END_REGION

REGION Network 24: +++++|MARCHA IZQUIERDA|+++++
   RUNG wire#powerrail
      Contact( #Cinta.Habilitado )
      Contact( #Cinta.Permiso.Izquierda )
      wire#w1
      Contact( #OkAlarma )
      Coil( #Cinta.Salidas.MarchaIzq )
   END_RUNG
   RUNG wire#powerrail
      I_Contact( #Cinta.Entradas.Auto )
   END_RUNG wire#w1
   // the same network as SCL:
   #Cinta.Salidas.MarchaIzq := ((#Cinta.Habilitado AND #Cinta.Permiso.Izquierda) OR NOT #Cinta.Entradas.Auto) AND #OkAlarma;
END_REGION

REGION Network 25: +++++|CINTA EN MARCHA|+++++
   RUNG wire#powerrail
      Contact( #Cinta.Salidas.MarchaAdelante )
      wire#w1
      Coil( #EnMarcha )
   END_RUNG
   RUNG wire#powerrail
      Contact( #Cinta.Salidas.MarchaAtras )
   END_RUNG wire#w1
   RUNG wire#powerrail
      Contact( #Cinta.Salidas.MarchaDch )
   END_RUNG wire#w1
   RUNG wire#powerrail
      Contact( #Cinta.Salidas.MarchaIzq )
   END_RUNG wire#w1
   // the same network as SCL:
   #EnMarcha := #Cinta.Salidas.MarchaAdelante OR #Cinta.Salidas.MarchaAtras OR #Cinta.Salidas.MarchaDch OR #Cinta.Salidas.MarchaIzq;
END_REGION

REGION Network 26: +++++|TIEMPO DE TRABAJO|+++++
   #Cinta."Timer"[1].TON(IN := #EnMarcha AND NOT #Cinta.TimerON[1], PT := T#1s);
   #Cinta.TimerON[1] := #Cinta."Timer"[1].Q;
   IF #Cinta."Timer"[1].Q THEN #Cinta.HMI.segTrabajo := #Cinta.HMI.segTrabajo + 1; END_IF;
   IF #EnMarcha AND (#Cinta.HMI.segTrabajo >= 60) THEN
       #Cinta.HMI.minTrabajo := #Cinta.HMI.minTrabajo + 1;
       #Cinta.HMI.segTrabajo := 0;
   END_IF;
   IF #EnMarcha AND (#Cinta.HMI.minTrabajo >= 60) THEN
       #Cinta.HMI.horaTrabajo := #Cinta.HMI.horaTrabajo + 1;
       #Cinta.HMI.minTrabajo := 0;
   END_IF;
END_REGION
END_FUNCTION

// folder: 01_E/S

FUNCTION "FC_ED" : Void   // FC2, LAD
{ S7_Optimized_Access := 'TRUE' }
VERSION : 0.1
BEGIN

REGION Network 1 (STL)

         A     "LAE-High";
         =     "ED"."LAE-High";

         A     "LAE-Low";
         =     "ED"."LAE-Low";

         A     "LAE-Pallet";
         =     "ED"."LAE-Pallet";

         A     "SLEN";
         =     "ED".SLEN;

         A     "SREN";
         =     "ED".SREN;

         A     "SREX";
         =     "ED".SREX;

         A     "SLEX";
         =     "ED".SLEX;

         A     "Marcha";
         =     "ED".Marcha;

         A     "Paro";
         =     "ED".Paro;

         A     "Reset";
         =     "ED".Reset;

         A     "Seta Emergencia";
         =     "ED"."Seta Emergencia";

         A     "SL";
         =     "ED".SL;

         A     "Manual";
         =     "ED".Manual;

         A     "Auto";
         =     "ED".Auto;
END_REGION
END_FUNCTION

FUNCTION "FC_SD" : Void   // FC3, LAD
{ S7_Optimized_Access := 'TRUE' }
VERSION : 0.1
BEGIN

REGION Network 1 (STL)
         A     "SD"."CT-right";
         =     "CT-right";

         A     "SD"."CT-left";
         =     "CT-left";

         A     "SD"."CT-Unload";
         =     "CT-Unload";

         A     "SD"."CT-Load";
         =     "CT-Load";

         A     "SD".CE;
         =     "CE";

         A     "SD".CL;
         =     "CL";

         A     "SD".CR;
         =     "CR";

         A     "SD".Emitter;
         =     "Emitter";

         A     "SD"."Remover left";
         =     "Remover left";

         A     "SD"."Remover right";
         =     "Remover right";

         A     "SD"."Start light";
         =     "Start light";

         A     "SD"."Stop light";
         =     "Stop light";

         A     "SD"."Reset light";
         =     "Reset light";
END_REGION
END_FUNCTION

// folder: 10_Zona de Clasificacion

FUNCTION "FC_ZonaClasificacion" : Void   // FC200, LAD
TITLE = +++++|CLASIFICACION CAJAS SEGUN TAMAÑO|+++++
{ S7_Optimized_Access := 'TRUE' }
VERSION : 0.1
// DERECHA = CAJAS GRANDES
// IZQUIERDA = CAJAS PEQUEÑAS
   VAR_TEMP   // added for the SCL form of the ladder/FBD networks
      _w1 : Bool;
      _w2 : Bool;
      _w3 : Bool;
      _w4 : Bool;
   END_VAR
BEGIN

REGION Network 1 (STL): +++++|TRATAMIENTO SENSORES|+++++
   //LAE HIGH
         CALL  "FC_SensorDigital"
         ( Sensor     := "ED"."LAE-High",
           Negado     := FALSE,
           Retardo    := 0,
           UDT_Sensor := "DB_SensoresDigitales"."LAE-High"
         );
   //LAE LOW
         CALL  "FC_SensorDigital"
         ( Sensor     := "ED"."LAE-Low",
           Negado     := FALSE,
           Retardo    := 0,
           UDT_Sensor := "DB_SensoresDigitales"."LAE-Low"
         );
   //LAE PALLET
         CALL  "FC_SensorDigital"
         ( Sensor     := "ED"."LAE-Pallet",
           Negado     := FALSE,
           Retardo    := 0,
           UDT_Sensor := "DB_SensoresDigitales"."LAE-Pallet"
         );
   //SLEN
         CALL  "FC_SensorDigital"
         ( Sensor     := "ED".SLEN,
           Negado     := TRUE,
           Retardo    := 0,
           UDT_Sensor := "DB_SensoresDigitales".SLEN
         );
   //SREN
         CALL  "FC_SensorDigital"
         ( Sensor     := "ED".SREN,
           Negado     := TRUE,
           Retardo    := 0,
           UDT_Sensor := "DB_SensoresDigitales".SREN
         );
   //SREX
         CALL  "FC_SensorDigital"
         ( Sensor     := "ED".SREX,
           Negado     := TRUE,
           Retardo    := 0,
           UDT_Sensor := "DB_SensoresDigitales".SREX
         );
   //SLEX
         CALL  "FC_SensorDigital"
         ( Sensor     := "ED".SLEX,
           Negado     := TRUE,
           Retardo    := 0,
           UDT_Sensor := "DB_SensoresDigitales".SLEX
         );
   //Seta de Emergencia
         CALL  "FC_SensorDigital"
         ( Sensor     := "ED"."Seta Emergencia",
           Negado     := TRUE,
           Retardo    := 0,
           UDT_Sensor := "DB_SensoresDigitales".SetaEmergencia
         );
   //SL
         CALL  "FC_SensorDigital"
         ( Sensor     := "ED".SL,
           Negado     := FALSE,
           Retardo    := 0,
           UDT_Sensor := "DB_SensoresDigitales".SL
         );
   //Paro
         CALL  "FC_SensorDigital"
         ( Sensor     := "ED".Paro,
           Negado     := TRUE,
           Retardo    := 0,
           UDT_Sensor := "DB_SensoresDigitales".Paro
         );
END_REGION

REGION Network 2 (STL): +++++|MARCHA / PARO|+++++
   //sistema en MARCHA

         A     "ED".Marcha;
         AN    "DB_SensoresDigitales".SetaEmergencia.Value;
         AN    "DB_SensoresDigitales".Paro.Value;
         S     "DB_ZonaClasificacion".EnMarcha;
         R     "DB_ZonaClasificacion".EnParo;

   //SISTEMA EN PARO

         A     "DB_SensoresDigitales".SetaEmergencia.Value;
         O     "DB_SensoresDigitales".Paro.Value;
         R     "DB_ZonaClasificacion".EnMarcha;
         S     "DB_ZonaClasificacion".EnParo;

   //LUCES DEL SISTEMA

         A     "DB_ZonaClasificacion".EnMarcha;
         =     "SD"."Start light";
   //ACTIVA LA LUZ VERDE CUANDO ESTE EN MARCHA
         A     "DB_ZonaClasificacion".EnParo;
         =     "SD"."Stop light";
   //ACTIVA LA LUZ ROJA CUANDO ESTE EN PARO
END_REGION

REGION Network 3 (SCL): +++++|LOGICA DE CONTROL|+++++
END_REGION

REGION Network 4: CAJA ESPERANDO EN ENTRADA CT
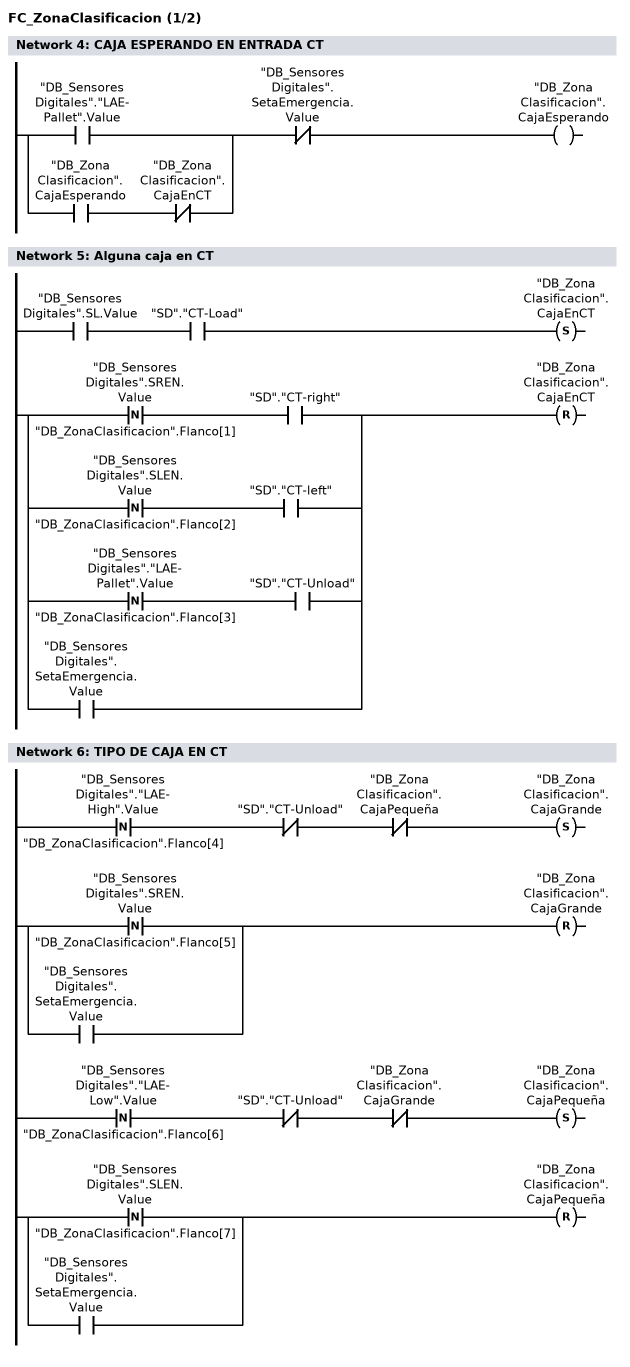
   RUNG wire#powerrail
      Contact( "DB_SensoresDigitales"."LAE-Pallet".Value )
      wire#w1
      I_Contact( "DB_SensoresDigitales".SetaEmergencia.Value )
      Coil( "DB_ZonaClasificacion".CajaEsperando )
   END_RUNG
   RUNG wire#powerrail
      Contact( "DB_ZonaClasificacion".CajaEsperando )
      I_Contact( "DB_ZonaClasificacion".CajaEnCT )
   END_RUNG wire#w1
   // the same network as SCL:
   "DB_ZonaClasificacion".CajaEsperando := ("DB_SensoresDigitales"."LAE-Pallet".Value OR ("DB_ZonaClasificacion".CajaEsperando AND NOT "DB_ZonaClasificacion".CajaEnCT)) AND NOT "DB_SensoresDigitales".SetaEmergencia.Value;
END_REGION

REGION Network 5: Alguna caja en CT
   RUNG wire#powerrail
      Contact( "DB_SensoresDigitales".SL.Value )
      Contact( "SD"."CT-Load" )
      S_Coil( "DB_ZonaClasificacion".CajaEnCT )
   END_RUNG
   RUNG wire#powerrail
      N_Contact(operand := "DB_SensoresDigitales".SREN.Value, bit := "DB_ZonaClasificacion".Flanco[1])
      Contact( "SD"."CT-right" )
      wire#w1
      R_Coil( "DB_ZonaClasificacion".CajaEnCT )
   END_RUNG
   RUNG wire#powerrail
      N_Contact(operand := "DB_SensoresDigitales".SLEN.Value, bit := "DB_ZonaClasificacion".Flanco[2])
      Contact( "SD"."CT-left" )
   END_RUNG wire#w1
   RUNG wire#powerrail
      N_Contact(operand := "DB_SensoresDigitales"."LAE-Pallet".Value, bit := "DB_ZonaClasificacion".Flanco[3])
      Contact( "SD"."CT-Unload" )
   END_RUNG wire#w1
   RUNG wire#powerrail
      Contact( "DB_SensoresDigitales".SetaEmergencia.Value )
   END_RUNG wire#w1
   // the same network as SCL:
   IF "DB_SensoresDigitales".SL.Value AND "SD"."CT-Load" THEN
       "DB_ZonaClasificacion".CajaEnCT := TRUE;
   END_IF;
   #_w1 := NOT "DB_SensoresDigitales".SREN.Value AND "DB_ZonaClasificacion".Flanco[1];   // falling edge of "DB_SensoresDigitales".SREN.Value
   "DB_ZonaClasificacion".Flanco[1] := "DB_SensoresDigitales".SREN.Value;
   #_w2 := NOT "DB_SensoresDigitales".SLEN.Value AND "DB_ZonaClasificacion".Flanco[2];   // falling edge of "DB_SensoresDigitales".SLEN.Value
   "DB_ZonaClasificacion".Flanco[2] := "DB_SensoresDigitales".SLEN.Value;
   #_w3 := NOT "DB_SensoresDigitales"."LAE-Pallet".Value AND "DB_ZonaClasificacion".Flanco[3];   // falling edge of "DB_SensoresDigitales"."LAE-Pallet".Value
   "DB_ZonaClasificacion".Flanco[3] := "DB_SensoresDigitales"."LAE-Pallet".Value;
   IF (#_w1 AND "SD"."CT-right") OR (#_w2 AND "SD"."CT-left") OR (#_w3 AND "SD"."CT-Unload") OR "DB_SensoresDigitales".SetaEmergencia.Value THEN
       "DB_ZonaClasificacion".CajaEnCT := FALSE;
   END_IF;
END_REGION

REGION Network 6: TIPO DE CAJA EN CT
   RUNG wire#powerrail
      N_Contact(operand := "DB_SensoresDigitales"."LAE-High".Value, bit := "DB_ZonaClasificacion".Flanco[4])
      I_Contact( "SD"."CT-Unload" )
      I_Contact( "DB_ZonaClasificacion".CajaPequeña )
      S_Coil( "DB_ZonaClasificacion".CajaGrande )
   END_RUNG
   RUNG wire#powerrail
      N_Contact(operand := "DB_SensoresDigitales".SREN.Value, bit := "DB_ZonaClasificacion".Flanco[5])
      wire#w1
      R_Coil( "DB_ZonaClasificacion".CajaGrande )
   END_RUNG
   RUNG wire#powerrail
      Contact( "DB_SensoresDigitales".SetaEmergencia.Value )
   END_RUNG wire#w1
   RUNG wire#powerrail
      N_Contact(operand := "DB_SensoresDigitales"."LAE-Low".Value, bit := "DB_ZonaClasificacion".Flanco[6])
      I_Contact( "SD"."CT-Unload" )
      I_Contact( "DB_ZonaClasificacion".CajaGrande )
      S_Coil( "DB_ZonaClasificacion".CajaPequeña )
   END_RUNG
   RUNG wire#powerrail
      N_Contact(operand := "DB_SensoresDigitales".SLEN.Value, bit := "DB_ZonaClasificacion".Flanco[7])
      wire#w2
      R_Coil( "DB_ZonaClasificacion".CajaPequeña )
   END_RUNG
   RUNG wire#powerrail
      Contact( "DB_SensoresDigitales".SetaEmergencia.Value )
   END_RUNG wire#w2
   // the same network as SCL:
   #_w1 := NOT "DB_SensoresDigitales"."LAE-High".Value AND "DB_ZonaClasificacion".Flanco[4];   // falling edge of "DB_SensoresDigitales"."LAE-High".Value
   "DB_ZonaClasificacion".Flanco[4] := "DB_SensoresDigitales"."LAE-High".Value;
   IF #_w1 AND NOT "SD"."CT-Unload" AND NOT "DB_ZonaClasificacion".CajaPequeña THEN
       "DB_ZonaClasificacion".CajaGrande := TRUE;
   END_IF;
   #_w2 := NOT "DB_SensoresDigitales".SREN.Value AND "DB_ZonaClasificacion".Flanco[5];   // falling edge of "DB_SensoresDigitales".SREN.Value
   "DB_ZonaClasificacion".Flanco[5] := "DB_SensoresDigitales".SREN.Value;
   IF #_w2 OR "DB_SensoresDigitales".SetaEmergencia.Value THEN
       "DB_ZonaClasificacion".CajaGrande := FALSE;
   END_IF;
   #_w3 := NOT "DB_SensoresDigitales"."LAE-Low".Value AND "DB_ZonaClasificacion".Flanco[6];   // falling edge of "DB_SensoresDigitales"."LAE-Low".Value
   "DB_ZonaClasificacion".Flanco[6] := "DB_SensoresDigitales"."LAE-Low".Value;
   IF #_w3 AND NOT "SD"."CT-Unload" AND NOT "DB_ZonaClasificacion".CajaGrande THEN
       "DB_ZonaClasificacion".CajaPequeña := TRUE;
   END_IF;
   #_w4 := NOT "DB_SensoresDigitales".SLEN.Value AND "DB_ZonaClasificacion".Flanco[7];   // falling edge of "DB_SensoresDigitales".SLEN.Value
   "DB_ZonaClasificacion".Flanco[7] := "DB_SensoresDigitales".SLEN.Value;
   IF #_w4 OR "DB_SensoresDigitales".SetaEmergencia.Value THEN
       "DB_ZonaClasificacion".CajaPequeña := FALSE;
   END_IF;
END_REGION

REGION Network 7: CAJAS EN CR
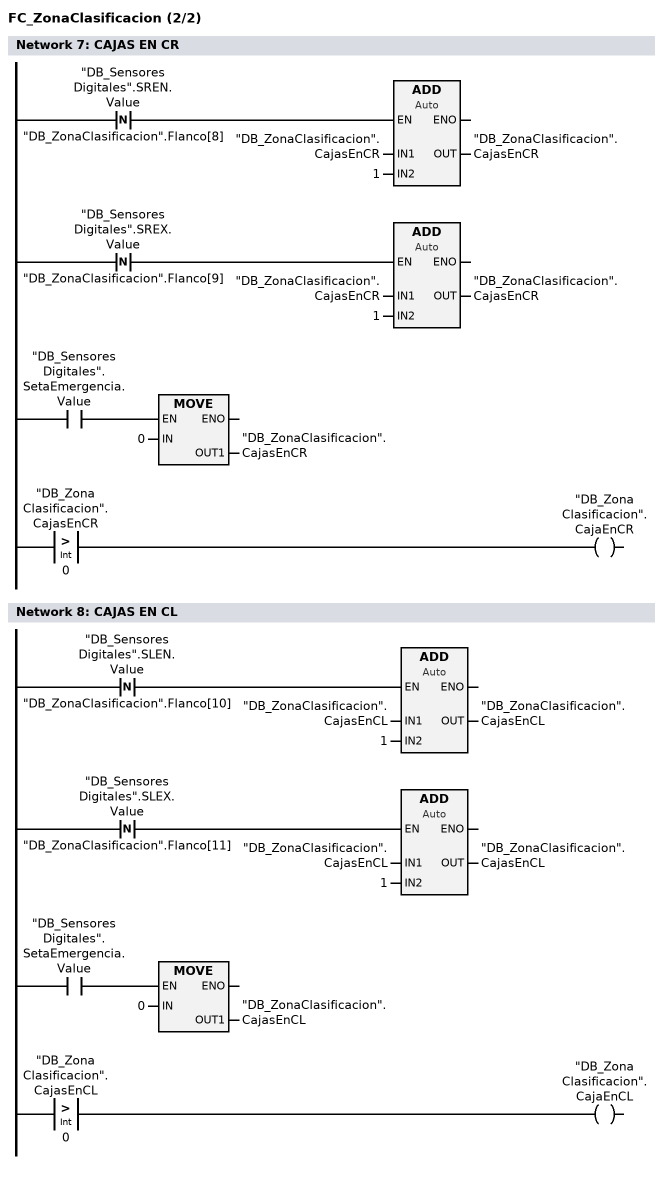
   RUNG wire#powerrail
      N_Contact(operand := "DB_SensoresDigitales".SREN.Value, bit := "DB_ZonaClasificacion".Flanco[8])
      Add(in1 := "DB_ZonaClasificacion".CajasEnCR, in2 := 1, out => "DB_ZonaClasificacion".CajasEnCR)
   END_RUNG
   RUNG wire#powerrail
      N_Contact(operand := "DB_SensoresDigitales".SREX.Value, bit := "DB_ZonaClasificacion".Flanco[9])
      Add(in1 := "DB_ZonaClasificacion".CajasEnCR, in2 := 1, out => "DB_ZonaClasificacion".CajasEnCR)
   END_RUNG
   RUNG wire#powerrail
      Contact( "DB_SensoresDigitales".SetaEmergencia.Value )
      Move(in := 0, out1 => "DB_ZonaClasificacion".CajasEnCR)
   END_RUNG
   RUNG wire#powerrail
      { S7_Templates := "SrcType := Int" } GT_Contact(in1 := "DB_ZonaClasificacion".CajasEnCR, in2 := 0)
      Coil( "DB_ZonaClasificacion".CajaEnCR )
   END_RUNG
   // the same network as SCL:
   #_w1 := NOT "DB_SensoresDigitales".SREN.Value AND "DB_ZonaClasificacion".Flanco[8];   // falling edge of "DB_SensoresDigitales".SREN.Value
   "DB_ZonaClasificacion".Flanco[8] := "DB_SensoresDigitales".SREN.Value;
   IF #_w1 THEN "DB_ZonaClasificacion".CajasEnCR := "DB_ZonaClasificacion".CajasEnCR + 1; END_IF;
   #_w2 := NOT "DB_SensoresDigitales".SREX.Value AND "DB_ZonaClasificacion".Flanco[9];   // falling edge of "DB_SensoresDigitales".SREX.Value
   "DB_ZonaClasificacion".Flanco[9] := "DB_SensoresDigitales".SREX.Value;
   IF #_w2 THEN "DB_ZonaClasificacion".CajasEnCR := "DB_ZonaClasificacion".CajasEnCR + 1; END_IF;
   IF "DB_SensoresDigitales".SetaEmergencia.Value THEN "DB_ZonaClasificacion".CajasEnCR := 0; END_IF;
   "DB_ZonaClasificacion".CajaEnCR := "DB_ZonaClasificacion".CajasEnCR > 0;
END_REGION

REGION Network 8: CAJAS EN CL
   RUNG wire#powerrail
      N_Contact(operand := "DB_SensoresDigitales".SLEN.Value, bit := "DB_ZonaClasificacion".Flanco[10])
      Add(in1 := "DB_ZonaClasificacion".CajasEnCL, in2 := 1, out => "DB_ZonaClasificacion".CajasEnCL)
   END_RUNG
   RUNG wire#powerrail
      N_Contact(operand := "DB_SensoresDigitales".SLEX.Value, bit := "DB_ZonaClasificacion".Flanco[11])
      Add(in1 := "DB_ZonaClasificacion".CajasEnCL, in2 := 1, out => "DB_ZonaClasificacion".CajasEnCL)
   END_RUNG
   RUNG wire#powerrail
      Contact( "DB_SensoresDigitales".SetaEmergencia.Value )
      Move(in := 0, out1 => "DB_ZonaClasificacion".CajasEnCL)
   END_RUNG
   RUNG wire#powerrail
      { S7_Templates := "SrcType := Int" } GT_Contact(in1 := "DB_ZonaClasificacion".CajasEnCL, in2 := 0)
      Coil( "DB_ZonaClasificacion".CajaEnCL )
   END_RUNG
   // the same network as SCL:
   #_w1 := NOT "DB_SensoresDigitales".SLEN.Value AND "DB_ZonaClasificacion".Flanco[10];   // falling edge of "DB_SensoresDigitales".SLEN.Value
   "DB_ZonaClasificacion".Flanco[10] := "DB_SensoresDigitales".SLEN.Value;
   IF #_w1 THEN "DB_ZonaClasificacion".CajasEnCL := "DB_ZonaClasificacion".CajasEnCL + 1; END_IF;
   #_w2 := NOT "DB_SensoresDigitales".SLEX.Value AND "DB_ZonaClasificacion".Flanco[11];   // falling edge of "DB_SensoresDigitales".SLEX.Value
   "DB_ZonaClasificacion".Flanco[11] := "DB_SensoresDigitales".SLEX.Value;
   IF #_w2 THEN "DB_ZonaClasificacion".CajasEnCL := "DB_ZonaClasificacion".CajasEnCL + 1; END_IF;
   IF "DB_SensoresDigitales".SetaEmergencia.Value THEN "DB_ZonaClasificacion".CajasEnCL := 0; END_IF;
   "DB_ZonaClasificacion".CajaEnCL := "DB_ZonaClasificacion".CajasEnCL > 0;
END_REGION

NETWORK
TITLE = +++++|CINTAS|+++++

NETWORK
TITLE = +++++|UNIDIRECCIONALES|+++++

REGION Network 11 (STL): CE
   //Habilitado por HMI
         A     "DB_Generalidades".SiempreON;
         =     "DB_Cintas".Unidireccional.CE.HMI.Habilitado;

   //AUTO REARMES

         A     "DB_Generalidades".SiempreON;
         =     "DB_Cintas".Unidireccional.CE.AutoRearme[1];
         =     "DB_Cintas".Unidireccional.CE.AutoRearme[2];
         =     "DB_Cintas".Unidireccional.CE.AutoRearme[3];
         =     "DB_Cintas".Unidireccional.CE.AutoRearme[4];
         =     "DB_Cintas".Unidireccional.CE.AutoRearme[5];

   //ENTRADAS

         A     "DB_Generalidades".SiempreOFF;
         =     "DB_Cintas".Unidireccional.CE.Entradas.Termico;
         =     "DB_Cintas".Unidireccional.CE.Entradas.Disyuntor;
         =     "DB_Cintas".Unidireccional.CE.Entradas.ConfMarcha;
         =     "DB_Cintas".Unidireccional.CE.Entradas.FalloVariador;

         A     "ED".Auto;
         AN    "ED".Manual;
         =     "DB_Cintas".Unidireccional.CE.Entradas.Auto;

         A     "DB_ZonaClasificacion".EnParo;
         =     "DB_Cintas".Unidireccional.CE.Entradas.ParoxSeguridad;

   //PERMISO EXTERNO

         A     "DB_ZonaClasificacion".EnMarcha;
         A(;
         AN    "DB_ZonaClasificacion".CajaEnCT;
         O(;
         A     "DB_ZonaClasificacion".CajaEnCT;
         AN    "DB_SensoresDigitales"."LAE-Pallet".Value;
         );
         );

         =     "DB_Cintas".Unidireccional.CE.Permiso.Externo;

   //LLAMADA CE

         CALL  "FC_Cinta"
         ( Cinta := "DB_Cintas".Unidireccional.CE
         );

   //SALIDAS

         A     "DB_Cintas".Unidireccional.CE.Salidas.Marcha;
         =     "SD".CE;
END_REGION

REGION Network 12 (STL): CR
   //Habilitado por HMI
         A     "DB_Generalidades".SiempreON;
         =     "DB_Cintas".Unidireccional.CR.HMI.Habilitado;

   //AUTO REARMES

         A     "DB_Generalidades".SiempreON;
         =     "DB_Cintas".Unidireccional.CR.AutoRearme[1];
         =     "DB_Cintas".Unidireccional.CR.AutoRearme[2];
         =     "DB_Cintas".Unidireccional.CR.AutoRearme[3];
         =     "DB_Cintas".Unidireccional.CR.AutoRearme[4];
         =     "DB_Cintas".Unidireccional.CR.AutoRearme[5];

   //ENTRADAS

         A     "DB_Generalidades".SiempreOFF;
         =     "DB_Cintas".Unidireccional.CR.Entradas.Termico;
         =     "DB_Cintas".Unidireccional.CR.Entradas.Disyuntor;
         =     "DB_Cintas".Unidireccional.CR.Entradas.ConfMarcha;
         =     "DB_Cintas".Unidireccional.CR.Entradas.FalloVariador;

         A     "ED".Auto;
         AN    "ED".Manual;
         =     "DB_Cintas".Unidireccional.CR.Entradas.Auto;

         A     "DB_ZonaClasificacion".EnParo;
         =     "DB_Cintas".Unidireccional.CR.Entradas.ParoxSeguridad;

   //PERMISO EXTERNO

         A     "DB_ZonaClasificacion".EnMarcha;
         A(;
         A     "SD"."CT-right";
         O     "DB_ZonaClasificacion".CajaEnCR;
         );
         =     "DB_Cintas".Unidireccional.CR.Permiso.Externo;

   //LLAMADA CR

         CALL  "FC_Cinta"
         ( Cinta := "DB_Cintas".Unidireccional.CR
         );

   //SALIDAS

         A     "DB_Cintas".Unidireccional.CR.Salidas.Marcha;
         =     "SD".CR;
END_REGION

REGION Network 13 (STL): CL
   //Habilitado por HMI
         A     "DB_Generalidades".SiempreON;
         =     "DB_Cintas".Unidireccional.CL.HMI.Habilitado;

   //AUTO REARMES

         A     "DB_Generalidades".SiempreON;
         =     "DB_Cintas".Unidireccional.CL.AutoRearme[1];
         =     "DB_Cintas".Unidireccional.CL.AutoRearme[2];
         =     "DB_Cintas".Unidireccional.CL.AutoRearme[3];
         =     "DB_Cintas".Unidireccional.CL.AutoRearme[4];
         =     "DB_Cintas".Unidireccional.CL.AutoRearme[5];

   //ENTRADAS

         A     "DB_Generalidades".SiempreOFF;
         =     "DB_Cintas".Unidireccional.CL.Entradas.Termico;
         =     "DB_Cintas".Unidireccional.CL.Entradas.Disyuntor;
         =     "DB_Cintas".Unidireccional.CL.Entradas.ConfMarcha;
         =     "DB_Cintas".Unidireccional.CL.Entradas.FalloVariador;

         A     "ED".Auto;
         AN    "ED".Manual;
         =     "DB_Cintas".Unidireccional.CL.Entradas.Auto;

         A     "DB_ZonaClasificacion".EnParo;
         =     "DB_Cintas".Unidireccional.CL.Entradas.ParoxSeguridad;

   //PERMISO EXTERNO

         A     "DB_ZonaClasificacion".EnMarcha;
         A(;
         A     "SD"."CT-left";
         O     "DB_ZonaClasificacion".CajaEnCL;
         );

         =     "DB_Cintas".Unidireccional.CL.Permiso.Externo;

   //LLAMADA CL

         CALL  "FC_Cinta"
         ( Cinta := "DB_Cintas".Unidireccional.CL
         );

   //SALIDAS

         A     "DB_Cintas".Unidireccional.CL.Salidas.Marcha;
         =     "SD".CL;
END_REGION

NETWORK
TITLE = +++++|BIDIRECCIONALES|+++++

REGION Network 15 (STL): CT
   //Habilitado por HMI
         A     "DB_Generalidades".SiempreON;
         =     "DB_Cintas".Bidireccional.CT.HMI.Habilitado;

   //AUTO REARMES

         A     "DB_Generalidades".SiempreON;
         =     "DB_Cintas".Bidireccional.CT.AutoRearme[1];
         =     "DB_Cintas".Bidireccional.CT.AutoRearme[2];
         =     "DB_Cintas".Bidireccional.CT.AutoRearme[3];
         =     "DB_Cintas".Bidireccional.CT.AutoRearme[4];
         =     "DB_Cintas".Bidireccional.CT.AutoRearme[5];

   //ENTRADAS

         A     "DB_Generalidades".SiempreOFF;
         =     "DB_Cintas".Bidireccional.CT.Entradas.Termico;
         =     "DB_Cintas".Bidireccional.CT.Entradas.Disyuntor;
         =     "DB_Cintas".Bidireccional.CT.Entradas.ConfMarcha;
         =     "DB_Cintas".Bidireccional.CT.Entradas.FalloVariador;

         A     "ED".Auto;
         AN    "ED".Manual;
         =     "DB_Cintas".Bidireccional.CT.Entradas.Auto;

         A     "DB_ZonaClasificacion".EnParo;
         =     "DB_Cintas".Bidireccional.CT.Entradas.ParoxSeguridad;

   //PERMISO EXTERNO

   //Permiso ADELANTE
         A     "DB_ZonaClasificacion".EnMarcha;
         A     "DB_ZonaClasificacion".CajaEsperando;
         AN    "DB_ZonaClasificacion".CajaEnCT;
         =     "DB_Cintas".Bidireccional.CT.Permiso.Adelante;

   //Permiso Derecha

         A     "DB_ZonaClasificacion".EnMarcha;
         A     "DB_ZonaClasificacion".CajaEnCT;
         A     "DB_ZonaClasificacion".CajaGrande;
         A(;
         AN    "DB_ZonaClasificacion".CajaEnCR;
         O(;
         A     "DB_ZonaClasificacion".CajaEnCR;
         A     "SD".CR;
         );
         );
         =     "DB_Cintas".Bidireccional.CT.Permiso.Derecha;

   //Permiso Izquierda

         A     "DB_ZonaClasificacion".EnMarcha;
         A     "DB_ZonaClasificacion".CajaEnCT;
         A     "DB_ZonaClasificacion".CajaPequeña;
         A(;
         AN    "DB_ZonaClasificacion".CajaEnCL;
         O(;
         A     "DB_ZonaClasificacion".CajaEnCL;
         A     "SD".CL;
         );
         );

         =     "DB_Cintas".Bidireccional.CT.Permiso.Izquierda;


   //LLAMADA CT

         CALL  "FC_Cinta_Bidireccional"
         ( Cinta := "DB_Cintas".Bidireccional.CT
         );

   //SALIDAS

         A     "DB_Cintas".Bidireccional.CT.Salidas.MarchaAtras;
         =     "SD"."CT-Unload";

         A     "DB_Cintas".Bidireccional.CT.Salidas.MarchaAdelante;
         =     "SD"."CT-Load";

         A     "DB_Cintas".Bidireccional.CT.Salidas.MarchaDch;
         =     "SD"."CT-right";

         A     "DB_Cintas".Bidireccional.CT.Salidas.MarchaIzq;
         =     "SD"."CT-left";
END_REGION
END_FUNCTION